INTERFACE IXtsTrack

PROPERTY TrackLength : mc_lreal
GET
END_GET
END_PROPERTY

END_INTERFACE

(* stored: Version 1.1.0.1, ProductVersion 3.1.4024.9
   Itf IXtsTrack: Id {82297094-0948-4f1a-ba6d-1d7e13cae51c}
   Property TrackLength: Id {ae84ce8b-979a-4af0-b89f-31b2e12cbe71}
   Get Get: Id {a37d7fd5-e1b9-4ae5-a693-7fa42723933b} *)
